PROGRAM MAIN
VAR
	Counter:	INT;
	Counter2:	CTU;
END_VAR

Counter := Counter + 1;

Counter2(CU := TRUE, PV := 10);

END_PROGRAM

(* stored: Version 1.1.0.1, ProductVersion 3.1.4024.11
   POU MAIN: Id {e01add17-90ea-4f25-ad6d-ba1fc3d88082}, SpecialFunc None *)
